// TwinCAT 3 PLC project MFX_BE_LENS_INTERLOCK
// ProgramVersion: 3.1.0.9
// libraries:
//   Tc2_Standard, * (Beckhoff Automation GmbH)
//   Tc2_System, * (Beckhoff Automation GmbH)
//   Tc3_Interfaces, * (Beckhoff Automation GmbH)
//   Tc3_Module, * (Beckhoff Automation GmbH)
//   Tc2_ModbusSrv,3.3.1.0,Beckhoff Automation GmbH
// project tree:
//   DUTs/ LENS.TcDUT, RADII_LIMIT.TcDUT, ST_FloatRange.TcDUT, ST_TableRow.TcDUT
//   / GlobalTextList.TcGTLO, PlcTask.TcTTO
//   GVLs/ GVL.TcGVL
//   POUs/ FB_EnergyTables.TcPOU, FB_LENS_SYSTEM.TcPOU, F_EFF_RADIUS.TcPOU, FB_HEARTBEAT.TcPOU (not stored), FB_LimitLookup.TcPOU, F_GetXRTLensIndex.TcPOU, MAIN.TcPOU, p_MPSSup.TcPOU, p_XLegacyPLCModbus.TcPOU (not stored)
//   POUs/Modbus/ p_ModbusRx_OutputCoils.TcPOU, p_ModbusRx_PLCMemory.TcPOU, p_ModbusTx_InputCoils.TcPOU, p_ModbusTx_InputReg.TcPOU, p_ModbusTx_OutputCoils.TcPOU, p_ModbusTx_PLCMemory.TcPOU
// real-time tasks:
//   TASK PlcTask: cycle T#10ms, priority 20, ADS port 350
// I/O:
//   DEVICE Device 2 (CX-BK)
//     Box 1 (CX-BK)
// variable links:
//   MFX_BE_LENS_INTERLOCK/MFX_BE_LENS_INTERLOCK Instance <-> Device 2 (CX-BK)/Box 1 (CX-BK)
//     PlcTask Outputs/GVL.bTRIP_MPS <-> Term 2 (KL2794)/Channel 1/Output

CONFIGURATION MFX_BE_LENS_INTERLOCK
    RESOURCE PLC ON TwinCAT3
        TASK PlcTask(INTERVAL := T#10ms, PRIORITY := 20);
        PROGRAM MAIN WITH PlcTask : MAIN;
    END_RESOURCE
END_CONFIGURATION

// ---- DUTs/LENS.TcDUT
TYPE LENS :
STRUCT
    IN     : BOOL; //Inserted state of the Lens
    KNOWN  : BOOL; //Whether state of Lens is definite
    RADIUS : REAL; //Current radius of lens
END_STRUCT
END_TYPE

// ---- DUTs/RADII_LIMIT.TcDUT
TYPE RADII_LIMIT :
STRUCT
    // Trip occurs when the effective radius falls inbetween TRIP_LOW and TRIP_HIGH (inclusive).
    TRIP_LOW  : REAL := 0;     // Trip effective radius low
    TRIP_HIGH : REAL := 10000; // Trip effective radius high
END_STRUCT
END_TYPE

// ---- DUTs/ST_FloatRange.TcDUT
TYPE ST_FloatRange :
STRUCT
    fLow  : REAL;
    fHigh : REAL;
END_STRUCT
END_TYPE

// ---- DUTs/ST_TableRow.TcDUT
TYPE ST_TableRow :
STRUCT
	fEnergy : LREAL;
    fLow  : LREAL;
    fHigh : LREAL;
END_STRUCT
END_TYPE

// ---- GVLs/GVL.TcGVL
VAR_GLOBAL
	(* Fault handling - inputs *)
    i_xFAULT_CLEAR    			: BOOL;  // Clear fault bit
	i_iUpdateRequestSeq			: DINT;  // Parameter update request sequence number

    (* Fault Handling - active faults *)
    bHeartbeatAlive     		: BOOL; // [Active] Whether heartbeat has updated
    bFAULT    AT %Q*    		: BOOL; // [Active] Whether Lens Interlock has tripped
    bStateFault	        		: BOOL; // [Active] Whether lens is in an unknown state
    bLimitSummaryFault			: BOOL; // [Active] Whether limit has been violated
    bTableLimitFault 			: BOOL;	// [Active] Energy/lens combination disallowed in table
    bMinEnergyFault 			: BOOL;	// [Active] Minimum energy not met
    bRequiresTransfocatorFault 	: BOOL; // [Active] Transfocator lens required to be inserted 

    (* Fault Handling - latched faults *)
	q_bHeartbeatLatch					: BOOL; // Latch: heartbeat fault
	q_bFaultLatch  						: BOOL; // Latch: summary for *any* fault
    q_bStateLatch 						: BOOL;	// Latch: motor state/position unknown 
    q_bLimitSummaryFaultLatch    		: BOOL; // Latch: Summary fault due to energy/lens combination
	q_bTableLimitFaultLatch 			: BOOL;	// Latch: Table disallowed range match
    q_bMinEnergyFaultLatch 				: BOOL; // Latch: Minimum energy not met
    q_bRequiresTransfocatorFaultLatch 	: BOOL; // Latch: Transfocator lens required to be inserted

	fbEnergyTables : FB_EnergyTables;
	
	(* Fault handling - MPS signals *)
    bTRIP_MPS AT %Q*    		: BOOL;  // [Active] Bit output to MPS (trip when LOW)
	
    (*Lens Information *)
    ////////////////////////////////
    XRT_LENSES : ARRAY[1..10] OF LENS; //Set of XRT Lenses
    TFS_LENSES : ARRAY[1..10] OF LENS; //Set of TFS Lenses
    XRT_RADIUS : REAL; //Current Radius of XRT lenses
    TFS_RADIUS : REAL; //Current Radius of TFS lenses
	
    XRT_LENS_SYSTEM : FB_LENS_SYSTEM;
    TFS_LENS_SYSTEM : FB_LENS_SYSTEM;

    (* Effective radius trip regions - per XRT lens configuration *)
    ////////////////////////////////////////////////////////////////
    NO_LENS_LIMIT : RADII_LIMIT;
    LENS1_LIMIT : RADII_LIMIT;
    LENS2_LIMIT : RADII_LIMIT;
    LENS3_LIMIT : RADII_LIMIT;	
	
	(* Feedback to the IOC *)
    q_stActiveLimit : RADII_LIMIT;
	
    fMinEnergies : ARRAY[0..3] OF LREAL;
    afbRequiresLensEnergyRange : ARRAY[0..3] OF ST_FloatRange;

    (* Heartbeat *)
    ////////////////////////////////
    i_xIOC_HEARTBEAT: BOOL; //Current status of heartbeat
    i_fPhotonEnergy : REAL; // Current photon energy (keep REAL for modbus compatibility)

    (* Modbus *)
    ///////////////////////////////
    LOTO_Override: BOOL := TRUE;
    /// test mb_Input_Coils[0] with "modpoll -r 32769 -t 1 127.0.0.1"
    mb_Input_Coils: ARRAY[0..255] OF BOOL;
    /// test mb_Output_Coils[0] with "modpoll -r 32769 -t 0 127.0.0.1"
    mb_Output_Coils: ARRAY[0..255] OF BOOL;
    /// test mb_Input_Registers[0] with "modpoll -r 32769 -t 3 127.0.0.1"
    mb_Input_Registers: ARRAY[0..255] OF WORD;
    /// test mb_Output_Registers[0] with "modpoll -r 32769 -t 4 127.0.0.1"
    mb_Output_Registers: ARRAY[0..255] OF WORD;
    /// test mb_PLC_Memory[0] with "modpoll -r 12289 -t 4 127.0.0.1"
    mb_PLC_Memory AT %MW0: ARRAY[0..1000] OF WORD;
	iCycleCount : WORD;

END_VAR

// ---- POUs/MAIN.TcPOU
PROGRAM MAIN
VAR
END_VAR

(* 16-bit cycle counter *)
iCycleCount := iCycleCount + 1;

fbEnergyTables();

(*  EPICS Rx UPDATE
    Modbus receive
*)
p_ModbusRx_OutputCoils();
p_ModbusRx_PLCMemory();
p_XLegacyPLCModbus();

(* Hard-code Lens Radii (microns) *)
XRT_LENSES[1].RADIUS := 750.0;
XRT_LENSES[2].RADIUS := 428.6;
XRT_LENSES[3].RADIUS := 333.3;

TFS_LENSES[1].RADIUS  := 0.0;   // A pinhole, not a lens.
TFS_LENSES[2].RADIUS  := 500.0;
TFS_LENSES[3].RADIUS  := 300.0;
TFS_LENSES[4].RADIUS  := 250.0;
TFS_LENSES[5].RADIUS  := 200.0;
TFS_LENSES[6].RADIUS  := 125.0;
TFS_LENSES[7].RADIUS  := 62.5;
TFS_LENSES[8].RADIUS  := 50.0;
TFS_LENSES[9].RADIUS  := 50.0;
TFS_LENSES[10].RADIUS := 50.0;

(* Additional trip settings

    Pre-focus 	Minimum energy [keV] 	Requires transfocator lens low [keV] 	Requires transfocator lens high [keV]
    NO_LENS 	0 	n/a 	n/a
    LENS3_333 	9.5 	9.5 	11.11
    LENS2_428 	8.28 	8.28 	10.02
    LENS1_750 	5.96 	5.96 	8.02

*)
fMinEnergies[0] := 0.0; (* No XRT lens *)
fMinEnergies[1] := 9500.0; (* XRT Lens 1 *)
fMinEnergies[2] := 8280.0; (* XRT lens 2 *)
fMinEnergies[3] := 5960.0; (* XRT lens 3 *)

afbRequiresLensEnergyRange[0].fLow := 0.0; (* No XRT lens / no restriction*)
afbRequiresLensEnergyRange[0].fHigh := 0.0;

afbRequiresLensEnergyRange[1].fLow := 9500.0; (* Lens 1: 9.5~11.11keV *)
afbRequiresLensEnergyRange[1].fHigh := 11110.0;

afbRequiresLensEnergyRange[2].fLow := 8280.0; (* Lens 2: 8.28 ~ 10.02 keV *)
afbRequiresLensEnergyRange[2].fHigh := 10020.0;

afbRequiresLensEnergyRange[3].fLow := 5960.0; (* Lens 3: 5.96 ~ 8.02 keV *)
afbRequiresLensEnergyRange[3].fHigh := 8020.0;

(*  MPS LOGIC SUMMARY *)
p_MPSSup();

(* 	EPICS Tx UPDATE
    Modbus Map Report
    IMPORTANT: This is the LAST subroutine to be called.
*)
p_ModbusTx_InputCoils();
p_ModbusTx_InputReg();
p_ModbusTx_PLCMemory();

END_PROGRAM

// ---- POUs/Modbus/p_ModbusRx_OutputCoils.TcPOU
PROGRAM p_ModbusRx_OutputCoils
VAR

END_VAR

//mb_Output_Coils[0];  //System Controls
//System Controls
//mb_Output_Coils[2];  //System Controls
//mb_Output_Coils[3];  //System Controls
//mb_Output_Coils[4];  //System Controls
//mb_Output_Coils[5];  //System Controls
//mb_Output_Coils[6];  //System Controls
//mb_Output_Coils[7];  //System Controls
//mb_Output_Coils[8];  //System Controls
//mb_Output_Coils[9];  //System Controls
TFS_LENSES[01].KNOWN:=TRUE;  //LOCKED OUT
TFS_LENSES[02].KNOWN:=mb_Output_Coils[11];  //Valve switch controls
TFS_LENSES[03].KNOWN:=mb_Output_Coils[12];  //Valve switch controls
TFS_LENSES[04].KNOWN:=mb_Output_Coils[13];  //Valve switch controls
TFS_LENSES[05].KNOWN:=mb_Output_Coils[14];  //Valve switch controls
TFS_LENSES[06].KNOWN:=mb_Output_Coils[15];  //Valve switch controls
TFS_LENSES[07].KNOWN:=mb_Output_Coils[16];  //Valve switch controls
TFS_LENSES[08].KNOWN:=mb_Output_Coils[17];  //Valve switch controls
TFS_LENSES[09].KNOWN:=mb_Output_Coils[18];  //Valve switch controls
TFS_LENSES[10].KNOWN:=mb_Output_Coils[19];  //Valve switch controls
XRT_LENSES[01].KNOWN:=mb_Output_Coils[20];
XRT_LENSES[02].KNOWN:=mb_Output_Coils[21];
XRT_LENSES[03].KNOWN:=mb_Output_Coils[22];
//mb_Output_Coils[23];  //Valve switch controls
//mb_Output_Coils[24];  //Valve switch controls
//mb_Output_Coils[25];  //Valve switch controls
//mb_Output_Coils[26];  //Valve switch controls
//mb_Output_Coils[27];  //Valve switch controls
//mb_Output_Coils[28];  //Valve switch controls
//mb_Output_Coils[29];  //Valve switch controls
TFS_LENSES[01].IN:=FALSE;  //Lockout
TFS_LENSES[02].IN:=mb_Output_Coils[31];  //Valve switch controls
TFS_LENSES[03].IN:=mb_Output_Coils[32];  //Valve switch controls
TFS_LENSES[04].IN:=mb_Output_Coils[33];  //Valve switch controls
TFS_LENSES[05].IN:=mb_Output_Coils[34];  //Valve switch controls
TFS_LENSES[06].IN:=mb_Output_Coils[35];  //Valve switch controls
TFS_LENSES[07].IN:=mb_Output_Coils[36];  //Valve switch controls
TFS_LENSES[08].IN:=mb_Output_Coils[37];  //Valve switch controls
TFS_LENSES[09].IN:=mb_Output_Coils[38];  //Valve switch controls
TFS_LENSES[10].IN:=mb_Output_Coils[39];  //Valve switch controls
XRT_LENSES[01].IN:=mb_Output_Coils[40];
XRT_LENSES[02].IN:=mb_Output_Coils[41];
XRT_LENSES[03].IN:=mb_Output_Coils[42];
//mb_Output_Coils[43];
//mb_Output_Coils[44];
//mb_Output_Coils[45];
//mb_Output_Coils[46];
//mb_Output_Coils[47];
//mb_Output_Coils[48];
//mb_Output_Coils[49];
i_xIOC_HEARTBEAT:=mb_Output_Coils[50];
i_xFAULT_CLEAR  :=mb_Output_Coils[51];
//mb_Output_Coils[52];  //Valve switch controls
//mb_Output_Coils[53];  //Valve switch controls
//mb_Output_Coils[54];  //Valve switch controls
//mb_Output_Coils[55];  //Valve switch controls
//mb_Output_Coils[56];  //Valve switch controls
//mb_Output_Coils[57];  //Valve switch controls
//mb_Output_Coils[58];  //Valve switch controls
//mb_Output_Coils[59];  //Valve switch controls
//mb_Output_Coils[60];  //Valve switch controls
//mb_Output_Coils[61];  //Valve switch controls
//mb_Output_Coils[62];  //Valve switch controls
//mb_Output_Coils[63];  //Valve switch controls
//mb_Output_Coils[64];  //Valve switch controls
//mb_Output_Coils[65];  //Valve switch controls
//mb_Output_Coils[66];  //Valve switch controls
//mb_Output_Coils[67];  //Valve switch controls
//mb_Output_Coils[68];  //Valve switch controls
//mb_Output_Coils[69];  //Valve switch controls
//mb_Output_Coils[70];  //Turbo Controls
//mb_Output_Coils[71];  //Turbo Controls
//mb_Output_Coils[72];  //Turbo Controls
//mb_Output_Coils[74];  //Turbo Controls
//mb_Output_Coils[75];  //Turbo Controls
//mb_Output_Coils[76];  //Turbo Controls
//mb_Output_Coils[77];  //Turbo Controls
//mb_Output_Coils[78];  //Turbo Controls
//mb_Output_Coils[79];  //Turbo Controls
//mb_Output_Coils[80];  //Turbo Controls
//mb_Output_Coils[81];  //Turbo Controls
//mb_Output_Coils[82];  //Turbo Controls
//mb_Output_Coils[83];  //Turbo Controls
//mb_Output_Coils[84];  //Turbo Controls
//mb_Output_Coils[85];  //Turbo Controls
//mb_Output_Coils[86];  //Turbo Controls
//mb_Output_Coils[87];  //Turbo Controls
//mb_Output_Coils[88];  //Turbo Controls
//mb_Output_Coils[89];  //Turbo Controls
//mb_Output_Coils[90];  //Turbo Controls
//mb_Output_Coils[91];  //Turbo Controls
//mb_Output_Coils[92];  //Turbo Controls
//mb_Output_Coils[93];  //Turbo Controls
//mb_Output_Coils[94];  //Turbo Controls
//mb_Output_Coils[95];  //Turbo Controls
//mb_Output_Coils[96];  //Turbo Controls
//mb_Output_Coils[97];  //Turbo Controls
//mb_Output_Coils[98];  //Turbo Controls
//mb_Output_Coils[99];  //Turbo Controls
//mb_Output_Coils[100];  //Turbo Controls
//mb_Output_Coils[101];  //Turbo Controls
//mb_Output_Coils[102];  //Turbo Controls
//mb_Output_Coils[103];  //Turbo Controls
//mb_Output_Coils[104];  //Turbo Controls
//mb_Output_Coils[105];  //Turbo Controls
//mb_Output_Coils[106];  //Turbo Controls
//mb_Output_Coils[107];  //Turbo Controls
//mb_Output_Coils[108];  //Turbo Controls
//mb_Output_Coils[109];  //Turbo Controls
//mb_Output_Coils[110];  //Turbo Controls
//mb_Output_Coils[111];  //Turbo Controls
//mb_Output_Coils[112];  //Turbo Controls
//mb_Output_Coils[113];  //Turbo Controls
//mb_Output_Coils[114];  //Turbo Controls
//mb_Output_Coils[115];  //Turbo Controls
//mb_Output_Coils[116];  //Turbo Controls
//mb_Output_Coils[117];  //Turbo Controls
//mb_Output_Coils[118];  //Turbo Controls
//mb_Output_Coils[119];  //Turbo Controls
//vgMXT_GCC_06.xHV_SW:=mb_Output_Coils[120];  //CC HV Enable
//vgDVD_GCC_02.xHV_SW:=mb_Output_Coils[121];  //CC HV Enable
//vgDVD_GCC_04.xHV_SW:=mb_Output_Coils[122];  //CC HV Enable
//vgMON_GCC_01.xHV_SW:=mb_Output_Coils[123];  //CC HV Enable
//vgDIA_GCC_01.xHV_SW:=mb_Output_Coils[124];  //CC HV Enable
//vgSB2_GCC_01.xHV_SW:=mb_Output_Coils[125];  //CC HV Enable
//vgDG1_GCC_01.xHV_SW:=mb_Output_Coils[126];  //CC HV Enable
//vgDG2_GCC_01.xHV_SW:=mb_Output_Coils[127];  //CC HV Enable
//mb_Output_Coils[128];  //CC HV Enable
//mb_Output_Coils[129];  //CC HV Enable
//mb_Output_Coils[130];  //CC HV Enable
//mb_Output_Coils[131];  //CC HV Enable
//mb_Output_Coils[132];  //CC HV Enable
//mb_Output_Coils[133];  //CC HV Enable
//mb_Output_Coils[134];  //CC HV Enable
//mb_Output_Coils[135];  //CC HV Enable
//mb_Output_Coils[136];  //CC HV Enable
//mb_Output_Coils[137];  //CC HV Enable
//mb_Output_Coils[138];  //CC HV Enable
//mb_Output_Coils[139];  //CC HV Enable
//mb_Output_Coils[140];  //CC HV Enable
//mb_Output_Coils[141];  //CC HV Enable
//mb_Output_Coils[142];  //CC HV Enable
//mb_Output_Coils[143];  //CC HV Enable
//mb_Output_Coils[144];  //CC HV Enable
//mb_Output_Coils[145];  //CC HV Enable
//mb_Output_Coils[146];  //CC HV Enable
//mb_Output_Coils[147];  //CC HV Enable
//mb_Output_Coils[148];  //CC HV Enable
//mb_Output_Coils[149];  //CC HV Enable
//mb_Output_Coils[150];  //CC HV Enable
//mb_Output_Coils[151];  //CC HV Enable
//mb_Output_Coils[152];  //CC HV Enable
//mb_Output_Coils[153];  //CC HV Enable
//mb_Output_Coils[154];  //CC HV Enable
//mb_Output_Coils[155];  //CC HV Enable
//mb_Output_Coils[156];  //CC HV Enable
//mb_Output_Coils[157];  //CC HV Enable
//mb_Output_Coils[158];  //CC HV Enable
//mb_Output_Coils[159];  //CC HV Enable
//mb_Output_Coils[160];  //
//mb_Output_Coils[161];  //
//mb_Output_Coils[162];  //
//mb_Output_Coils[163];  //
//mb_Output_Coils[164];  //
//mb_Output_Coils[165];  //
//mb_Output_Coils[166];  //
//mb_Output_Coils[167];  //
//mb_Output_Coils[168];  //
//mb_Output_Coils[169];  //
//mb_Output_Coils[170];  //
//mb_Output_Coils[171];  //
//mb_Output_Coils[172];  //
//mb_Output_Coils[173];  //
//mb_Output_Coils[174];  //
//mb_Output_Coils[175];  //
//mb_Output_Coils[176];  //
//mb_Output_Coils[177];  //
//mb_Output_Coils[178];  //
//mb_Output_Coils[179];  //
//mb_Output_Coils[180];  //
//mb_Output_Coils[181];  //
//mb_Output_Coils[182];  //
//mb_Output_Coils[183];  //
//mb_Output_Coils[184];  //
//mb_Output_Coils[185];  //
//mb_Output_Coils[186];  //
//mb_Output_Coils[187];  //
//mb_Output_Coils[188];  //
//mb_Output_Coils[189];  //
//mb_Output_Coils[190];  //
//mb_Output_Coils[191];  //
//mb_Output_Coils[192];  //
//mb_Output_Coils[193];  //
//mb_Output_Coils[194];  //
//mb_Output_Coils[195];  //
//mb_Output_Coils[196];  //
//mb_Output_Coils[197];  //
//mb_Output_Coils[198];  //
//mb_Output_Coils[199];  //
//mb_Output_Coils[200];  //Valve overrides
//mb_Output_Coils[201];  //Valve overrides
//mb_Output_Coils[202];  //Valve overrides
//mb_Output_Coils[203];  //Valve overrides
//mb_Output_Coils[204];  //
//mb_Output_Coils[205];  //
//mb_Output_Coils[206];  //
//mb_Output_Coils[207];  //
//mb_Output_Coils[208];  //
//mb_Output_Coils[209];  //
//mb_Output_Coils[210];  //
//mb_Output_Coils[211];  //
//mb_Output_Coils[212];  //
//mb_Output_Coils[213];  //
//mb_Output_Coils[214];  //
//mb_Output_Coils[215];  //
//mb_Output_Coils[216];  //
//mb_Output_Coils[217];  //
//mb_Output_Coils[218];  //
//mb_Output_Coils[219];  //
//mb_Output_Coils[220];  //
//mb_Output_Coils[221];  //
//mb_Output_Coils[222];  //
//mb_Output_Coils[223];  //
//mb_Output_Coils[224];  //
//mb_Output_Coils[225];  //
//mb_Output_Coils[226];  //
//mb_Output_Coils[227];  //
//mb_Output_Coils[228];  //
//mb_Output_Coils[229];  //
//mb_Output_Coils[230];  //
//mb_Output_Coils[231];  //
//mb_Output_Coils[232];  //
//mb_Output_Coils[233];  //
//mb_Output_Coils[234];  //
//mb_Output_Coils[235];  //
//mb_Output_Coils[236];  //
//mb_Output_Coils[237];  //
//mb_Output_Coils[238];  //
//mb_Output_Coils[239];  //
//mb_Output_Coils[240];  //
//mb_Output_Coils[241];  //
//mb_Output_Coils[242];  //
//mb_Output_Coils[243];  //
//mb_Output_Coils[244];  //
//mb_Output_Coils[245];  //
//mb_Output_Coils[246];  //
//mb_Output_Coils[247];  //
//mb_Output_Coils[248];  //
//mb_Output_Coils[249];  //
//mb_Output_Coils[250];  //
//mb_Output_Coils[251];  //
//mb_Output_Coils[252];  //
//mb_Output_Coils[253];  //
//mb_Output_Coils[254];  //
//mb_Output_Coils[255];  //

END_PROGRAM

// ---- POUs/Modbus/p_ModbusRx_PLCMemory.TcPOU
PROGRAM p_ModbusRx_PLCMemory
VAR
END_VAR

(*
{"MFX:LENS:",  "XRT_ONLY:LOW" , "aoFLOAT_PORT",    "0", "FLOAT32_LE",  "1", "1000",  "0", "um"}
{"MFX:LENS:",  "XRT_ONLY:HIGH", "aoFLOAT_PORT",    "2", "FLOAT32_LE",  "1", "1000",  "0", "um"}
{"MFX:LENS:", "LENS1_750:LOW" , "aoFLOAT_PORT",    "4", "FLOAT32_LE",  "1", "1000",  "0", "um"}
{"MFX:LENS:", "LENS1_750:HIGH", "aoFLOAT_PORT",    "6", "FLOAT32_LE",  "1", "1000",  "0", "um"}
{"MFX:LENS:", "LENS2_428:LOW" , "aoFLOAT_PORT",    "8", "FLOAT32_LE",  "1", "1000",  "0", "um"}
{"MFX:LENS:", "LENS2_428:HIGH", "aoFLOAT_PORT",   "10", "FLOAT32_LE",  "1", "1000",  "0", "um"}
{"MFX:LENS:", "LENS3_333:LOW" , "aoFLOAT_PORT",   "12", "FLOAT32_LE",  "1", "1000",  "0", "um"}
{"MFX:LENS:", "LENS3_333:HIGH", "aoFLOAT_PORT",   "14", "FLOAT32_LE",  "1", "1000",  "0", "um"}
*)
MEMCPY(srcAddr:=ADR(mb_PLC_Memory[ 0]), destAddr:=ADR(NO_LENS_LIMIT.TRIP_LOW), n:=SIZEOF(NO_LENS_LIMIT.TRIP_LOW));
MEMCPY(srcAddr:=ADR(mb_PLC_Memory[ 2]), destAddr:=ADR(NO_LENS_LIMIT.TRIP_HIGH), n:=SIZEOF(NO_LENS_LIMIT.TRIP_HIGH));

MEMCPY(srcAddr:=ADR(mb_PLC_Memory[ 4]), destAddr:=ADR(LENS1_LIMIT.TRIP_LOW), n:=SIZEOF(LENS1_LIMIT.TRIP_LOW));
MEMCPY(srcAddr:=ADR(mb_PLC_Memory[ 6]), destAddr:=ADR(LENS1_LIMIT.TRIP_HIGH), n:=SIZEOF(LENS1_LIMIT.TRIP_HIGH));

MEMCPY(srcAddr:=ADR(mb_PLC_Memory[ 8]), destAddr:=ADR(LENS2_LIMIT.TRIP_LOW), n:=SIZEOF(LENS2_LIMIT.TRIP_LOW));
MEMCPY(srcAddr:=ADR(mb_PLC_Memory[10]), destAddr:=ADR(LENS2_LIMIT.TRIP_HIGH), n:=SIZEOF(LENS2_LIMIT.TRIP_HIGH));

MEMCPY(srcAddr:=ADR(mb_PLC_Memory[12]), destAddr:=ADR(LENS3_LIMIT.TRIP_LOW), n:=SIZEOF(LENS3_LIMIT.TRIP_LOW));
MEMCPY(srcAddr:=ADR(mb_PLC_Memory[14]), destAddr:=ADR(LENS3_LIMIT.TRIP_HIGH), n:=SIZEOF(LENS3_LIMIT.TRIP_HIGH));

MEMCPY(srcAddr:=ADR(mb_PLC_Memory[16]), destAddr:=ADR(i_fPhotonEnergy), n:=SIZEOF(i_fPhotonEnergy));

MEMCPY(srcAddr:=ADR(mb_PLC_Memory[18]), destAddr:=ADR(i_iUpdateRequestSeq), n:=SIZEOF(i_iUpdateRequestSeq));

END_PROGRAM

// ---- POUs/p_MPSSup.TcPOU
PROGRAM p_MPSSup
VAR
    BEAT: FB_HEARTBEAT;
	fbHeartbeatLatch : RS;
	fbFaultLatch : RS;
    fbStateLatch : RS;
    fbLimitLatch : RS;
    fbTableLimitFaultLatch : RS;
    fbMinEnergyFaultLatch : RS;
    fbRequiresTransfocatorFaultLatch : RS;
	rtUpdate : R_TRIG;
	iLastSeq : DINT;
	bUpdateRequest: BOOL;
	
    LIMIT_FAULT : BOOL;

    fEnergyMin : LREAL;
    fRequiresTransfocatorEnergyLow : LREAL;
    fRequiresTransfocatorEnergyHigh : LREAL;
	fTripLow : LREAL;
	fTripHigh : LREAL;
	bEnergyInTable : BOOL;
	
    iLensIdx: INT;
	fbLimitLookup : FB_LimitLookup;

END_VAR

// Latch fault state
////////////////////

fbFaultLatch(SET:=bFAULT, RESET1:=i_xFAULT_CLEAR);
q_bFaultLatch := fbFaultLatch.Q1;

fbHeartbeatLatch(SET:=NOT bHeartbeatAlive, RESET1:=i_xFAULT_CLEAR);
q_bHeartbeatLatch := fbHeartbeatLatch.Q1;

fbStateLatch(SET:=bStateFault, RESET1:=i_xFAULT_CLEAR);
q_bStateLatch := fbStateLatch.Q1;

fbLimitLatch(SET:=bLimitSummaryFault, RESET1:=i_xFAULT_CLEAR);
q_bLimitSummaryFaultLatch := fbLimitLatch.Q1;

fbTableLimitFaultLatch(SET:=bTableLimitFault, RESET1:=i_xFAULT_CLEAR);
q_bTableLimitFaultLatch := fbTableLimitFaultLatch.Q1;

fbMinEnergyFaultLatch(SET:=bMinEnergyFault, RESET1:=i_xFAULT_CLEAR);
q_bMinEnergyFaultLatch := fbMinEnergyFaultLatch.Q1;

fbRequiresTransfocatorFaultLatch(SET:=bRequiresTransfocatorFault, RESET1:=i_xFAULT_CLEAR);
q_bRequiresTransfocatorFaultLatch := fbRequiresTransfocatorFaultLatch.Q1;

//IOC Heartbeat:
BEAT(BEAT:=i_xIOC_HEARTBEAT, DEADTIME:=TIME#0.5S);
bHeartbeatAlive := BEAT.ALIVE;

//XRT LENS SYSTEM
///////////////////////////
XRT_LENS_SYSTEM(LENSES:=XRT_LENSES, COUNT:=3);
XRT_RADIUS := XRT_LENS_SYSTEM.EFF_RADII; (* Propagated to EPICS *)

//TFS LENS SYSTEM
///////////////////////////
TFS_LENS_SYSTEM(LENSES:=TFS_LENSES, COUNT:=10);
TFS_RADIUS := TFS_LENS_SYSTEM.EFF_RADII; (* Propagated to EPICS *)

(* Reset our tracking variables *)
bTableLimitFault := FALSE;
bMinEnergyFault := FALSE;
bRequiresTransfocatorFault := FALSE;

(* Determine which XRT lens is inserted, and pick the correct range based on it. *)

IF NOT XRT_LENS_SYSTEM.UNKNOWN_FAULT THEN
	iLensIdx := F_GetXRTLensIndex();
	fbLimitLookup(
		fEnergy:=i_fPhotonEnergy,
		fLow=>fTripLow,
		fHigh=>fTripHigh,
		bEnergyInTable=>bEnergyInTable
	);

	q_stActiveLimit.TRIP_LOW := LREAL_TO_REAL(fTripLow);
	q_stActiveLimit.TRIP_HIGH := LREAL_TO_REAL(fTripHigh);

	IF bEnergyInTable AND fTripHigh > fTripLow THEN
		// Lens inserted and trip region specified:
		bTableLimitFault := (fTripLow <= TFS_RADIUS AND TFS_RADIUS <= fTripHigh);
	END_IF
	
	fEnergyMin := fMinEnergies[iLensIdx];
	fRequiresTransfocatorEnergyLow := afbRequiresLensEnergyRange[iLensIdx].fLow;
	fRequiresTransfocatorEnergyHigh := afbRequiresLensEnergyRange[iLensIdx].fHigh;
	
	(*
	Regardless of transfocator setting, the minimum energy must be
	greater than or equal to that shown in the table (Minimum energy [keV]).
	Trip if below.
	*)
	bMinEnergyFault := i_fPhotonEnergy < fEnergyMin;

	(*
	When a pre-focusing lens is inserted, there exists a range of photon
	energies in which at least one transfocator lens must be inserted.
	If the current photon energy is within this (inclusive) range and no
	lens is inserted, trip.
	*)
	IF fRequiresTransfocatorEnergyHigh > fRequiresTransfocatorEnergyLow THEN
		(* Check that we're in the given photon energy range *)
		IF fRequiresTransfocatorEnergyLow <= i_fPhotonEnergy AND i_fPhotonEnergy <= fRequiresTransfocatorEnergyHigh THEN
			(* And if so, trip when IN_COUNT == 0 *)
			bRequiresTransfocatorFault := (TFS_LENS_SYSTEM.IN_COUNT < 1);
		END_IF
	END_IF

END_IF

//Summarize faults
///////////////////////////

bLimitSummaryFault := (
	bTableLimitFault OR         // Inside the table-defined trip range
	bMinEnergyFault OR			// Below minimum required energy for XRT lens
	bRequiresTransfocatorFault	// Require transfocator lens in this range
);

//State Violations
bStateFault := (
	XRT_LENS_SYSTEM.UNKNOWN_FAULT OR  // XRT lens state unknown
	TFS_LENS_SYSTEM.UNKNOWN_FAULT OR  // Transfocator lens state unknown
	XRT_LENS_SYSTEM.IN_COUNT > 1      // Unexpected lens count
);

//Final Summary

// MPS trips when *LOW*. 
// 	So: bTRIP_MPS (False) when bFAULT (True)
// 	And bTRIP_MPS (True) when bFAULT (False)
bFAULT := bLimitSummaryFault OR bStateFault OR NOT bHeartbeatAlive;
bTRIP_MPS := NOT bFAULT;

(******************************)
(******************************)
(******************************)
(******************************)
bTRIP_MPS := TRUE; (* TEMPORARY: Alex requested the PLC never trip MPS for his overnight experiments *)
(* TODO: reviewers, this needs to be removed *)
(******************************)
(******************************)
(******************************)
(******************************)

END_PROGRAM

// ---- POUs/FB_LimitLookup.TcPOU
FUNCTION_BLOCK FB_LimitLookup
VAR_INPUT
	fEnergy : LREAL;
END_VAR
VAR_OUTPUT
	bEnergyInTable : BOOL;
	fLow : LREAL;
	fHigh : LREAL;
END_VAR
VAR
	(* TC version doesn't appear to support dynamic arrays here *)
	(* falling back to pointer-handling; sorry! *)
	stRow : POINTER TO ST_TableRow;
	stNextRow : POINTER TO ST_TableRow;
	iRowCount : UINT;
	iRowIdx : UINT;
	fSlope : LREAL;
	fEnergyDelta : LREAL;
	iLensIdx: INT;
END_VAR

iLensIdx := F_GetXRTLensIndex();

IF iLensIdx = 1 THEN
	stRow := ADR(fbEnergyTables.stLENS1_750);
	iRowCount := SIZEOF(fbEnergyTables.stLENS1_750) / SIZEOF(ST_TableRow);
ELSIF iLensIdx = 2 THEN
	stRow := ADR(fbEnergyTables.stLENS2_428);
	iRowCount := SIZEOF(fbEnergyTables.stLENS2_428) / SIZEOF(ST_TableRow);
ELSIF iLensIdx = 3 THEN
	stRow := ADR(fbEnergyTables.stLENS3_333);
	iRowCount := SIZEOF(fbEnergyTables.stLENS3_333) / SIZEOF(ST_TableRow);
ELSE
	stRow := ADR(fbEnergyTables.stNO_LENS);
	iRowCount := SIZEOF(fbEnergyTables.stNO_LENS) / SIZEOF(ST_TableRow);
END_IF

fLow := 0.0;
fHigh := 0.0;
bEnergyInTable := FALSE;

IF fEnergy < stRow^.fEnergy THEN
	RETURN;
END_IF

FOR iRowIdx := 0 TO iRowCount - 2
DO
(*
 result->energy = find_energy;
 double slope = (rows[upper_idx].low - rows[lower_idx].low) / delta_energy;
 result->low = rows[lower_idx].low + slope * (find_energy - rows[lower_idx].energy);

 slope = (rows[upper_idx].high - rows[lower_idx].high) / delta_energy;
 result->high = rows[lower_idx].high + slope * (find_energy - rows[lower_idx].energy);
*)
	stNextRow := ADR(stRow[1]);
	IF fEnergy >= stRow^.fEnergy AND fEnergy <= stNextRow^.fEnergy THEN
		fEnergyDelta := stNextRow^.fEnergy - stRow^.fEnergy;
		IF fEnergyDelta > 0.0 THEN
			bEnergyInTable := TRUE;
			// Interpolate between the points
			fSlope := (stNextRow^.fLow - stRow^.fLow) / fEnergyDelta;
			fLow := stRow^.fLow + fSlope * (fEnergy - stRow^.fEnergy);

			fSlope := (stNextRow^.fHigh - stRow^.fHigh) / fEnergyDelta;
			fHigh := stRow^.fHigh + fSlope * (fEnergy - stRow^.fEnergy);
		END_IF	
		RETURN;
	END_IF
	stRow := stNextRow;
END_FOR

END_FUNCTION_BLOCK

// ---- POUs/F_GetXRTLensIndex.TcPOU
FUNCTION F_GetXRTLensIndex : INT
VAR_INPUT
END_VAR
VAR
END_VAR

IF XRT_LENS_SYSTEM.LENSES[1].IN THEN
	F_GetXRTLensIndex := 1;
ELSIF XRT_LENS_SYSTEM.LENSES[2].IN THEN
	F_GetXRTLensIndex := 2;
ELSIF XRT_LENS_SYSTEM.LENSES[3].IN THEN
	F_GetXRTLensIndex := 3;
ELSE
	F_GetXRTLensIndex := 0;
END_IF

END_FUNCTION

// ---- POUs/Modbus/p_ModbusTx_InputCoils.TcPOU
PROGRAM p_ModbusTx_InputCoils
VAR
END_VAR
VAR_OUTPUT
END_VAR

(** NOTE: These values are mirrored in PLC memory output as well. **)
(** From an EPICS client perspective, it's easier to keep the data
    in synchronization when sent in one packet. The IOC now uses
    those values and these are vestigial for now.
**)


(* Online/active values *)
mb_Input_Coils[0]:=bHeartbeatAlive;
mb_Input_Coils[1]:=bFAULT;
mb_Input_Coils[2]:=bStateFault;
mb_Input_Coils[3]:=bLimitSummaryFault;
mb_Input_Coils[4]:=bMinEnergyFault;
mb_Input_Coils[5]:=bRequiresTransfocatorFault;
mb_Input_Coils[6]:=bTableLimitFault;
mb_Input_Coils[7]:=FALSE;
mb_Input_Coils[8]:=FALSE;
mb_Input_Coils[9]:=FALSE;

(* Latched fault information *)
mb_Input_Coils[10]:=q_bHeartbeatLatch;
mb_Input_Coils[11]:=q_bFaultLatch;
mb_Input_Coils[12]:=q_bStateLatch;
mb_Input_Coils[13]:=q_bLimitSummaryFaultLatch;
mb_Input_Coils[14]:=q_bMinEnergyFaultLatch;
mb_Input_Coils[15]:=q_bRequiresTransfocatorFaultLatch;
mb_Input_Coils[16]:=q_bTableLimitFaultLatch;
mb_Input_Coils[17]:=FALSE;
mb_Input_Coils[18]:=FALSE;
mb_Input_Coils[19]:=FALSE;

mb_Input_Coils[20]:=FALSE;  //Valve position readbacks
mb_Input_Coils[21]:=FALSE;  //Valve position readbacks
mb_Input_Coils[22]:=FALSE;  //Valve position readbacks
mb_Input_Coils[23]:=FALSE;  //Valve position readbacks
mb_Input_Coils[24]:=FALSE;  //Valve position readbacks
mb_Input_Coils[25]:=FALSE;  //Valve position readbacks
mb_Input_Coils[26]:=FALSE;  //Valve position readbacks
mb_Input_Coils[27]:=FALSE;  //Valve position readbacks
mb_Input_Coils[28]:=FALSE;  //Valve position readbacks
mb_Input_Coils[29]:=FALSE;  //Valve position readbacks
mb_Input_Coils[30]:=FALSE;  //Valve position readbacks
mb_Input_Coils[31]:=FALSE;  //Valve position readbacks
mb_Input_Coils[32]:=FALSE;  //Valve position readbacks
mb_Input_Coils[33]:=FALSE;  //Valve position readbacks
mb_Input_Coils[34]:=FALSE;  //Valve position readbacks
mb_Input_Coils[35]:=FALSE;  //Valve position readbacks
mb_Input_Coils[36]:=FALSE;  //Valve position readbacks
mb_Input_Coils[37]:=FALSE;  //Valve position readbacks
mb_Input_Coils[38]:=FALSE;  //Valve position readbacks
mb_Input_Coils[39]:=FALSE;  //Valve position readbacks
mb_Input_Coils[40]:=FALSE;  //Valve position readbacks
mb_Input_Coils[41]:=FALSE;  //Valve position readbacks
mb_Input_Coils[42]:=FALSE;  //Valve position readbacks
mb_Input_Coils[43]:=FALSE;  //Valve position readbacks
mb_Input_Coils[44]:=FALSE;  //Valve position readbacks
mb_Input_Coils[45]:=FALSE;  //Valve position readbacks
mb_Input_Coils[46]:=FALSE;  //Valve position readbacks
mb_Input_Coils[47]:=FALSE;  //Valve position readbacks
mb_Input_Coils[48]:=FALSE;  //Valve position readbacks
mb_Input_Coils[49]:=FALSE;  //Valve position readbacks
mb_Input_Coils[50]:=FALSE;  //Valve position readbacks
mb_Input_Coils[51]:=FALSE;  //Valve position readbacks
mb_Input_Coils[52]:=FALSE;  //Valve position readbacks
mb_Input_Coils[53]:=FALSE;  //Valve position readbacks
mb_Input_Coils[54]:=FALSE;  //Valve position readbacks
mb_Input_Coils[55]:=FALSE;  //Valve position readbacks
mb_Input_Coils[56]:=FALSE;  //Valve position readbacks
mb_Input_Coils[57]:=FALSE;  //Valve position readbacks
mb_Input_Coils[58]:=FALSE;  //Valve position readbacks
mb_Input_Coils[59]:=FALSE;  //Valve position readbacks
mb_Input_Coils[60]:=FALSE;  //Valve position readbacks
mb_Input_Coils[61]:=FALSE;  //Valve position readbacks
mb_Input_Coils[62]:=FALSE;  //Valve position readbacks
mb_Input_Coils[63]:=FALSE;  //Valve position readbacks
mb_Input_Coils[64]:=FALSE;  //Valve position readbacks
mb_Input_Coils[65]:=FALSE;  //Valve position readbacks
mb_Input_Coils[66]:=FALSE;  //Valve position readbacks
mb_Input_Coils[67]:=FALSE;  //Valve position readbacks
mb_Input_Coils[68]:=FALSE;  //Valve position readbacks
mb_Input_Coils[69]:=FALSE;  //Valve position readbacks
mb_Input_Coils[70]:=FALSE;  //Valve position readbacks
mb_Input_Coils[71]:=FALSE;  //Valve position readbacks
mb_Input_Coils[72]:=FALSE;  //Valve position readbacks
mb_Input_Coils[73]:=FALSE;  //Valve position readbacks
mb_Input_Coils[74]:=FALSE;  //Valve position readbacks
mb_Input_Coils[75]:=FALSE;  //Valve position readbacks
mb_Input_Coils[76]:=FALSE;  //Valve position readbacks
mb_Input_Coils[77]:=FALSE;  //Valve position readbacks
mb_Input_Coils[78]:=FALSE;  //Valve position readbacks
mb_Input_Coils[79]:=FALSE;  //Valve position readbacks
mb_Input_Coils[80]:=FALSE;  //Valve position readbacks
mb_Input_Coils[81]:=FALSE;  //Valve position readbacks
mb_Input_Coils[82]:=FALSE;  //Valve position readbacks
mb_Input_Coils[83]:=FALSE;  //Valve position readbacks
mb_Input_Coils[84]:=FALSE;  //Valve position readbacks
mb_Input_Coils[85]:=FALSE;  //Valve position readbacks
mb_Input_Coils[86]:=FALSE;  //Valve position readbacks
mb_Input_Coils[87]:=FALSE;  //Valve position readbacks
mb_Input_Coils[88]:=FALSE;  //Valve position readbacks
mb_Input_Coils[89]:=FALSE;  //Valve position readbacks
mb_Input_Coils[90]:=FALSE;  //Valve position readbacks
mb_Input_Coils[91]:=FALSE;  //Valve position readbacks
mb_Input_Coils[92]:=FALSE;  //Valve position readbacks
mb_Input_Coils[93]:=FALSE;  //Valve position readbacks
mb_Input_Coils[94]:=FALSE;  //Valve position readbacks
mb_Input_Coils[95]:=FALSE;  //Valve position readbacks
mb_Input_Coils[96]:=FALSE;  //Valve position readbacks
mb_Input_Coils[97]:=FALSE;  //Valve position readbacks
mb_Input_Coils[98]:=FALSE;  //Valve position readbacks
mb_Input_Coils[99]:=FALSE;  //Valve position readbacks
mb_Input_Coils[100]:=FALSE;  //Valve position readbacks
mb_Input_Coils[101]:=FALSE;  //Valve position readbacks
mb_Input_Coils[102]:=FALSE;  //Valve position readbacks
mb_Input_Coils[103]:=FALSE;  //Valve position readbacks
mb_Input_Coils[104]:=FALSE;  //Valve position readbacks
mb_Input_Coils[105]:=FALSE;  //Valve position readbacks
mb_Input_Coils[106]:=FALSE;  //Valve position readbacks
mb_Input_Coils[107]:=FALSE;  //Valve position readbacks
mb_Input_Coils[108]:=FALSE;  //Valve position readbacks
mb_Input_Coils[109]:=FALSE;  //Valve position readbacks
mb_Input_Coils[110]:=FALSE;  //Valve position readbacks
mb_Input_Coils[111]:=FALSE;  //Valve position readbacks
mb_Input_Coils[112]:=FALSE;  //Valve position readbacks
mb_Input_Coils[113]:=FALSE;  //Valve position readbacks
mb_Input_Coils[114]:=FALSE;  //Valve position readbacks
mb_Input_Coils[115]:=FALSE;  //Valve position readbacks
mb_Input_Coils[116]:=FALSE;  //Valve position readbacks
mb_Input_Coils[117]:=FALSE;  //Valve position readbacks
mb_Input_Coils[118]:=FALSE;  //Valve position readbacks
mb_Input_Coils[119]:=FALSE;  //Valve position readbacks
mb_Input_Coils[120]:=FALSE;  //Turbo pump readbacks
mb_Input_Coils[121]:=FALSE;  //Turbo pump readbacks
mb_Input_Coils[122]:=FALSE;  //Turbo pump readbacks
mb_Input_Coils[123]:=FALSE;  //Turbo pump readbacks
mb_Input_Coils[124]:=FALSE;  //Turbo pump readbacks
mb_Input_Coils[125]:=FALSE;  //Turbo pump readbacks
mb_Input_Coils[126]:=FALSE;  //Turbo pump readbacks
mb_Input_Coils[127]:=FALSE;  //Turbo pump readbacks
mb_Input_Coils[128]:=FALSE;  //Turbo pump readbacks
mb_Input_Coils[129]:=FALSE;  //Turbo pump readbacks
mb_Input_Coils[130]:=FALSE;  //Turbo pump readbacks
mb_Input_Coils[131]:=FALSE;  //Turbo pump readbacks
mb_Input_Coils[132]:=FALSE;  //Turbo pump readbacks
mb_Input_Coils[133]:=FALSE;  //Turbo pump readbacks
mb_Input_Coils[134]:=FALSE;  //Turbo pump readbacks
mb_Input_Coils[135]:=FALSE;  //Turbo pump readbacks
mb_Input_Coils[136]:=FALSE;  //Turbo pump readbacks
mb_Input_Coils[137]:=FALSE;  //Turbo pump readbacks
mb_Input_Coils[138]:=FALSE;  //Turbo pump readbacks
mb_Input_Coils[139]:=FALSE;  //Turbo pump readbacks
mb_Input_Coils[140]:=FALSE;  //Turbo pump readbacks
mb_Input_Coils[141]:=FALSE;  //Turbo pump readbacks
mb_Input_Coils[142]:=FALSE;  //Turbo pump readbacks
mb_Input_Coils[143]:=FALSE;  //Turbo pump readbacks
mb_Input_Coils[144]:=FALSE;  //Turbo pump readbacks
mb_Input_Coils[145]:=FALSE;  //Turbo pump readbacks
mb_Input_Coils[146]:=FALSE;  //Turbo pump readbacks
mb_Input_Coils[147]:=FALSE;  //Turbo pump readbacks
mb_Input_Coils[148]:=FALSE;  //Turbo pump readbacks
mb_Input_Coils[149]:=FALSE;  //Turbo pump readbacks
mb_Input_Coils[150]:=FALSE;  //Turbo pump readbacks
mb_Input_Coils[151]:=FALSE;  //Turbo pump readbacks
mb_Input_Coils[152]:=FALSE;  //Turbo pump readbacks
mb_Input_Coils[153]:=FALSE;  //Turbo pump readbacks
mb_Input_Coils[154]:=FALSE;  //Turbo pump readbacks
mb_Input_Coils[155]:=FALSE;  //Turbo pump readbacks
mb_Input_Coils[156]:=FALSE;  //Turbo pump readbacks
mb_Input_Coils[157]:=FALSE;  //Turbo pump readbacks
mb_Input_Coils[158]:=FALSE;  //Turbo pump readbacks
mb_Input_Coils[159]:=FALSE;  //Turbo pump readbacks
mb_Input_Coils[160]:=FALSE;  //Turbo pump readbacks
mb_Input_Coils[161]:=FALSE;  //Turbo pump readbacks
mb_Input_Coils[162]:=FALSE;  //Turbo pump readbacks
mb_Input_Coils[163]:=FALSE;  //Turbo pump readbacks
mb_Input_Coils[164]:=FALSE;  //Turbo pump readbacks
mb_Input_Coils[165]:=FALSE;  //Turbo pump readbacks
mb_Input_Coils[166]:=FALSE;  //Turbo pump readbacks
mb_Input_Coils[167]:=FALSE;  //Turbo pump readbacks
mb_Input_Coils[168]:=FALSE;  //Turbo pump readbacks
mb_Input_Coils[169]:=FALSE;  //Turbo pump readbacks
mb_Input_Coils[170]:=FALSE;  //Turbo pump readbacks
mb_Input_Coils[171]:=FALSE;  //Turbo pump readbacks
mb_Input_Coils[172]:=FALSE;  //Turbo pump readbacks
mb_Input_Coils[173]:=FALSE;  //Turbo pump readbacks
mb_Input_Coils[174]:=FALSE;  //Turbo pump readbacks
mb_Input_Coils[175]:=FALSE;  //Turbo pump readbacks
mb_Input_Coils[176]:=FALSE;  //Turbo pump readbacks
mb_Input_Coils[177]:=FALSE;  //Turbo pump readbacks
mb_Input_Coils[178]:=FALSE;  //Turbo pump readbacks
mb_Input_Coils[179]:=FALSE;  //Turbo pump readbacks
mb_Input_Coils[180]:=FALSE;  //Turbo pump readbacks
mb_Input_Coils[181]:=FALSE;  //Turbo pump readbacks
mb_Input_Coils[182]:=FALSE;  //Turbo pump readbacks
mb_Input_Coils[183]:=FALSE;  //Turbo pump readbacks
mb_Input_Coils[184]:=FALSE;  //Turbo pump readbacks
mb_Input_Coils[185]:=FALSE;  //Turbo pump readbacks
mb_Input_Coils[186]:=FALSE;  //Turbo pump readbacks
mb_Input_Coils[187]:=FALSE;  //Turbo pump readbacks
mb_Input_Coils[188]:=FALSE;  //Turbo pump readbacks
mb_Input_Coils[189]:=FALSE;  //Turbo pump readbacks
mb_Input_Coils[190]:=FALSE;  //Turbo pump readbacks
mb_Input_Coils[191]:=FALSE;  //Turbo pump readbacks
mb_Input_Coils[192]:=FALSE;  //Turbo pump readbacks
mb_Input_Coils[193]:=FALSE;  //Turbo pump readbacks
mb_Input_Coils[194]:=FALSE;  //Turbo pump readbacks
mb_Input_Coils[195]:=FALSE;  //Turbo pump readbacks
mb_Input_Coils[196]:=FALSE;  //Turbo pump readbacks
mb_Input_Coils[197]:=FALSE;  //Turbo pump readbacks
mb_Input_Coils[198]:=FALSE;  //Turbo pump readbacks
mb_Input_Coils[199]:=FALSE;  //Turbo pump readbacks
mb_Input_Coils[200]:=FALSE;  //Turbo pump readbacks
mb_Input_Coils[201]:=FALSE;  //Turbo pump readbacks
mb_Input_Coils[202]:=FALSE;  //Turbo pump readbacks
mb_Input_Coils[203]:=FALSE;  //Turbo pump readbacks
mb_Input_Coils[204]:=FALSE;  //Turbo pump readbacks
mb_Input_Coils[205]:=FALSE;  //Turbo pump readbacks
mb_Input_Coils[206]:=FALSE;  //Turbo pump readbacks
mb_Input_Coils[207]:=FALSE;  //Turbo pump readbacks
mb_Input_Coils[208]:=FALSE;  //Turbo pump readbacks
mb_Input_Coils[209]:=FALSE;  //Turbo pump readbacks
mb_Input_Coils[210]:=FALSE;  //Turbo pump readbacks
mb_Input_Coils[211]:=FALSE;  //Turbo pump readbacks
mb_Input_Coils[212]:=FALSE;  //Turbo pump readbacks
mb_Input_Coils[213]:=FALSE;  //Turbo pump readbacks
mb_Input_Coils[214]:=FALSE;  //Turbo pump readbacks
mb_Input_Coils[215]:=FALSE;  //Turbo pump readbacks
mb_Input_Coils[216]:=FALSE;  //Turbo pump readbacks
mb_Input_Coils[217]:=FALSE;  //Turbo pump readbacks
mb_Input_Coils[218]:=FALSE;  //Turbo pump readbacks
mb_Input_Coils[219]:=FALSE;  //Turbo pump readbacks
mb_Input_Coils[220]:=FALSE;  //VG readbacks
mb_Input_Coils[221]:=FALSE;  //VG readbacks
mb_Input_Coils[222]:=FALSE;  //VG readbacks
mb_Input_Coils[223]:=FALSE;  //VG readbacks
mb_Input_Coils[224]:=FALSE;  //VG readbacks
mb_Input_Coils[225]:=FALSE;  //VG readbacks
mb_Input_Coils[226]:=FALSE;  //VG readbacks
mb_Input_Coils[227]:=FALSE;  //VG readbacks
mb_Input_Coils[228]:=FALSE;  //VG readbacks
mb_Input_Coils[229]:=FALSE;  //VG readbacks
mb_Input_Coils[230]:=FALSE;  //VG readbacks
mb_Input_Coils[231]:=FALSE;  //VG readbacks
mb_Input_Coils[232]:=FALSE;  //VG readbacks
mb_Input_Coils[233]:=FALSE;  //VG readbacks
mb_Input_Coils[234]:=FALSE;  //VG readbacks
mb_Input_Coils[235]:=FALSE;  //VG readbacks
mb_Input_Coils[236]:=FALSE;  //VG readbacks
mb_Input_Coils[237]:=FALSE;  //VG readbacks
mb_Input_Coils[238]:=FALSE;  //VG readbacks
mb_Input_Coils[239]:=FALSE;  //VG readbacks
mb_Input_Coils[240]:=FALSE;  //VG readbacks
mb_Input_Coils[241]:=FALSE;  //VG readbacks
mb_Input_Coils[242]:=FALSE;  //VG readbacks
mb_Input_Coils[243]:=FALSE;  //VG readbacks
mb_Input_Coils[244]:=FALSE;  //VG readbacks
mb_Input_Coils[245]:=FALSE;  //VG readbacks
mb_Input_Coils[246]:=FALSE;  //VG readbacks
mb_Input_Coils[247]:=FALSE;  //VG readbacks
mb_Input_Coils[248]:=FALSE;  //VG readbacks
mb_Input_Coils[249]:=FALSE;  //VG readbacks
mb_Input_Coils[250]:=FALSE;  //VG readbacks
mb_Input_Coils[251]:=FALSE;  //VG readbacks
mb_Input_Coils[252]:=FALSE;  //VG readbacks
mb_Input_Coils[253]:=FALSE;  //VG readbacks
mb_Input_Coils[254]:=FALSE;  //VG readbacks
mb_Input_Coils[255]:=FALSE;  //VG readbacks

END_PROGRAM

// ---- POUs/Modbus/p_ModbusTx_InputReg.TcPOU
PROGRAM p_ModbusTx_InputReg
VAR

END_VAR

mb_Input_Registers[0]:=0;  //System info
mb_Input_Registers[1]:=0;  //System info
mb_Input_Registers[2]:=0;  //System info
mb_Input_Registers[3]:=0;  //System info
mb_Input_Registers[4]:=0;  //System info
mb_Input_Registers[5]:=0;  //System info
mb_Input_Registers[6]:=0;  //System info
mb_Input_Registers[7]:=0;  //System info
mb_Input_Registers[8]:=0;  //System info
mb_Input_Registers[9]:=0;  //System info
mb_Input_Registers[10]:=0;  //VG pressure readbacks
mb_Input_Registers[11]:=0;  //VG pressure readbacks
mb_Input_Registers[12]:=0;  //VG pressure readbacks
mb_Input_Registers[13]:=0;  //VG pressure readbacks
mb_Input_Registers[14]:=0;  //VG pressure readbacks
mb_Input_Registers[15]:=0;  //VG pressure readbacks
mb_Input_Registers[16]:=0;  //VG pressure readbacks
mb_Input_Registers[17]:=0;  //VG pressure readbacks
mb_Input_Registers[18]:=0;  //VG pressure readbacks
mb_Input_Registers[19]:=0;  //VG pressure readbacks
mb_Input_Registers[20]:=0;  //VG pressure readbacks
mb_Input_Registers[21]:=0;  //VG pressure readbacks
mb_Input_Registers[22]:=0;  //VG pressure readbacks
mb_Input_Registers[23]:=0;  //VG pressure readbacks
mb_Input_Registers[24]:=0;  //VG pressure readbacks
mb_Input_Registers[25]:=0;  //VG pressure readbacks
mb_Input_Registers[26]:=0;  //VG pressure readbacks
mb_Input_Registers[27]:=0;  //VG pressure readbacks
mb_Input_Registers[28]:=0;  //VG pressure readbacks
mb_Input_Registers[29]:=0;  //VG pressure readbacks
mb_Input_Registers[30]:=0;  //VG pressure readbacks
mb_Input_Registers[31]:=0;  //VG pressure readbacks
mb_Input_Registers[32]:=0;  //VG pressure readbacks
mb_Input_Registers[33]:=0;  //VG pressure readbacks
mb_Input_Registers[34]:=0;  //VG pressure readbacks
mb_Input_Registers[35]:=0;  //VG pressure readbacks
mb_Input_Registers[36]:=0;  //VG pressure readbacks
mb_Input_Registers[37]:=0;  //VG pressure readbacks
mb_Input_Registers[38]:=0;  //VG pressure readbacks
mb_Input_Registers[39]:=0;  //VG pressure readbacks
mb_Input_Registers[40]:=0;  //VG pressure readbacks
mb_Input_Registers[41]:=0;  //VG pressure readbacks
mb_Input_Registers[42]:=0;  //VG pressure readbacks
mb_Input_Registers[43]:=0;  //VG pressure readbacks
mb_Input_Registers[44]:=0;  //VG pressure readbacks
mb_Input_Registers[45]:=0;  //VG pressure readbacks
mb_Input_Registers[46]:=0;  //VG pressure readbacks
mb_Input_Registers[47]:=0;  //VG pressure readbacks
mb_Input_Registers[48]:=0;  //VG pressure readbacks
mb_Input_Registers[49]:=0;  //VG pressure readbacks
mb_Input_Registers[50]:=0;  //VG pressure readbacks
mb_Input_Registers[51]:=0;  //VG pressure readbacks
mb_Input_Registers[52]:=0;  //VG pressure readbacks
mb_Input_Registers[53]:=0;  //VG pressure readbacks
mb_Input_Registers[54]:=0;  //VG pressure readbacks
mb_Input_Registers[55]:=0;  //VG pressure readbacks
mb_Input_Registers[56]:=0;  //VG pressure readbacks
mb_Input_Registers[57]:=0;  //VG pressure readbacks
mb_Input_Registers[58]:=0;  //VG pressure readbacks
mb_Input_Registers[59]:=0;  //VG pressure readbacks
mb_Input_Registers[60]:=0;  //VG pressure readbacks
mb_Input_Registers[61]:=0;  //VG pressure readbacks
mb_Input_Registers[62]:=0;  //VG pressure readbacks
mb_Input_Registers[63]:=0;  //VG pressure readbacks
mb_Input_Registers[64]:=0;  //VG pressure readbacks
mb_Input_Registers[65]:=0;  //VG pressure readbacks
mb_Input_Registers[66]:=0;  //VG pressure readbacks
mb_Input_Registers[67]:=0;  //VG pressure readbacks
mb_Input_Registers[68]:=0;  //VG pressure readbacks
mb_Input_Registers[69]:=0;  //VG pressure readbacks
mb_Input_Registers[70]:=0;  //VG state readbacks
mb_Input_Registers[71]:=0;  //VG state readbacks
mb_Input_Registers[72]:=0;  //VG state readbacks
mb_Input_Registers[73]:=0;  //VG state readbacks
mb_Input_Registers[74]:=0;  //VG state readbacks
mb_Input_Registers[75]:=0;  //VG state readbacks
mb_Input_Registers[76]:=0;  //VG state readbacks
mb_Input_Registers[77]:=0;  //VG state readbacks
mb_Input_Registers[78]:=0;  //VG state readbacks
mb_Input_Registers[79]:=0;  //VG state readbacks
mb_Input_Registers[80]:=0;  //VG state readbacks
mb_Input_Registers[81]:=0;  //VG state readbacks
mb_Input_Registers[82]:=0;  //VG state readbacks
mb_Input_Registers[83]:=0;  //VG state readbacks
mb_Input_Registers[84]:=0;  //VG state readbacks
mb_Input_Registers[85]:=0;  //VG state readbacks
mb_Input_Registers[86]:=0;  //VG state readbacks
mb_Input_Registers[87]:=0;  //VG state readbacks
mb_Input_Registers[88]:=0;  //VG state readbacks
mb_Input_Registers[89]:=0;  //VG state readbacks
mb_Input_Registers[90]:=0;  //VG state readbacks
mb_Input_Registers[91]:=0;  //VG state readbacks
mb_Input_Registers[92]:=0;  //VG state readbacks
mb_Input_Registers[93]:=0;  //VG state readbacks
mb_Input_Registers[94]:=0;  //VG state readbacks
mb_Input_Registers[95]:=0;  //VG state readbacks
mb_Input_Registers[96]:=0;  //VG state readbacks
mb_Input_Registers[97]:=0;  //VG state readbacks
mb_Input_Registers[98]:=0;  //VG state readbacks
mb_Input_Registers[99]:=0;  //VG state readbacks
mb_Input_Registers[100]:=0;  //VG state readbacks
mb_Input_Registers[101]:=0;  //VG state readbacks
mb_Input_Registers[102]:=0;  //VG state readbacks
mb_Input_Registers[103]:=0;  //VG state readbacks
mb_Input_Registers[104]:=0;  //VG state readbacks
mb_Input_Registers[105]:=0;  //VG state readbacks
mb_Input_Registers[106]:=0;  //VG state readbacks
mb_Input_Registers[107]:=0;  //VG state readbacks
mb_Input_Registers[108]:=0;  //VG state readbacks
mb_Input_Registers[109]:=0;  //VG state readbacks
mb_Input_Registers[110]:=0;  //VG state readbacks
mb_Input_Registers[111]:=0;  //VG state readbacks
mb_Input_Registers[112]:=0;  //VG state readbacks
mb_Input_Registers[113]:=0;  //VG state readbacks
mb_Input_Registers[114]:=0;  //VG state readbacks
mb_Input_Registers[115]:=0;  //VG state readbacks
mb_Input_Registers[116]:=0;  //VG state readbacks
mb_Input_Registers[117]:=0;  //VG state readbacks
mb_Input_Registers[118]:=0;  //VG state readbacks
mb_Input_Registers[119]:=0;  //VG state readbacks
mb_Input_Registers[120]:=0;  //default
mb_Input_Registers[121]:=0;  //default
mb_Input_Registers[122]:=0;  //default
mb_Input_Registers[123]:=0;  //default
mb_Input_Registers[124]:=0;  //default
mb_Input_Registers[125]:=0;  //default
mb_Input_Registers[126]:=0;  //default
mb_Input_Registers[127]:=0;  //default
mb_Input_Registers[128]:=0;  //default
mb_Input_Registers[129]:=0;  //default
mb_Input_Registers[130]:=0;  //default
mb_Input_Registers[131]:=0;  //default
mb_Input_Registers[132]:=0;  //default
mb_Input_Registers[133]:=0;  //default
mb_Input_Registers[134]:=0;  //default
mb_Input_Registers[135]:=0;  //default
mb_Input_Registers[136]:=0;  //default
mb_Input_Registers[137]:=0;  //default
mb_Input_Registers[138]:=0;  //default
mb_Input_Registers[139]:=0;  //default
mb_Input_Registers[140]:=0;  //default
mb_Input_Registers[141]:=0;  //default
mb_Input_Registers[142]:=0;  //default
mb_Input_Registers[143]:=0;  //default
mb_Input_Registers[144]:=0;  //default
mb_Input_Registers[145]:=0;  //default
mb_Input_Registers[146]:=0;  //default
mb_Input_Registers[147]:=0;  //default
mb_Input_Registers[148]:=0;  //default
mb_Input_Registers[149]:=0;  //default
mb_Input_Registers[150]:=0;  //default
mb_Input_Registers[151]:=0;  //default
mb_Input_Registers[152]:=0;  //default
mb_Input_Registers[153]:=0;  //default
mb_Input_Registers[154]:=0;  //default
mb_Input_Registers[155]:=0;  //default
mb_Input_Registers[156]:=0;  //default
mb_Input_Registers[157]:=0;  //default
mb_Input_Registers[158]:=0;  //default
mb_Input_Registers[159]:=0;  //default
mb_Input_Registers[160]:=0;  //default
mb_Input_Registers[161]:=0;  //default
mb_Input_Registers[162]:=0;  //default
mb_Input_Registers[163]:=0;  //default
mb_Input_Registers[164]:=0;  //default
mb_Input_Registers[165]:=0;  //default
mb_Input_Registers[166]:=0;  //default
mb_Input_Registers[167]:=0;  //default
mb_Input_Registers[168]:=0;  //default
mb_Input_Registers[169]:=0;  //default
mb_Input_Registers[170]:=0;  //default
mb_Input_Registers[171]:=0;  //default
mb_Input_Registers[172]:=0;  //default
mb_Input_Registers[173]:=0;  //default
mb_Input_Registers[174]:=0;  //default
mb_Input_Registers[175]:=0;  //default
mb_Input_Registers[176]:=0;  //default
mb_Input_Registers[177]:=0;  //default
mb_Input_Registers[178]:=0;  //default
mb_Input_Registers[179]:=0;  //default
mb_Input_Registers[180]:=0;  //default
mb_Input_Registers[181]:=0;  //default
mb_Input_Registers[182]:=0;  //default
mb_Input_Registers[183]:=0;  //default
mb_Input_Registers[184]:=0;  //default
mb_Input_Registers[185]:=0;  //default
mb_Input_Registers[186]:=0;  //default
mb_Input_Registers[187]:=0;  //default
mb_Input_Registers[188]:=0;  //default
mb_Input_Registers[189]:=0;  //default
mb_Input_Registers[190]:=0;  //default
mb_Input_Registers[191]:=0;  //default
mb_Input_Registers[192]:=0;  //default
mb_Input_Registers[193]:=0;  //default
mb_Input_Registers[194]:=0;  //default
mb_Input_Registers[195]:=0;  //default
mb_Input_Registers[196]:=0;  //default
mb_Input_Registers[197]:=0;  //default
mb_Input_Registers[198]:=0;  //default
mb_Input_Registers[199]:=0;  //default
mb_Input_Registers[200]:=0;  //default
mb_Input_Registers[201]:=0;  //default
mb_Input_Registers[202]:=0;  //default
mb_Input_Registers[203]:=0;  //default
mb_Input_Registers[204]:=0;  //default
mb_Input_Registers[205]:=0;  //default
mb_Input_Registers[206]:=0;  //default
mb_Input_Registers[207]:=0;  //default
mb_Input_Registers[208]:=0;  //default
mb_Input_Registers[209]:=0;  //default
mb_Input_Registers[210]:=0;  //default
mb_Input_Registers[211]:=0;  //default
mb_Input_Registers[212]:=0;  //default
mb_Input_Registers[213]:=0;  //default
mb_Input_Registers[214]:=0;  //default
mb_Input_Registers[215]:=0;  //default
mb_Input_Registers[216]:=0;  //default
mb_Input_Registers[217]:=0;  //default
mb_Input_Registers[218]:=0;  //default
mb_Input_Registers[219]:=0;  //default
mb_Input_Registers[220]:=0;  //default
mb_Input_Registers[221]:=0;  //default
mb_Input_Registers[222]:=0;  //default
mb_Input_Registers[223]:=0;  //default
mb_Input_Registers[224]:=0;  //default
mb_Input_Registers[225]:=0;  //default
mb_Input_Registers[226]:=0;  //default
mb_Input_Registers[227]:=0;  //default
mb_Input_Registers[228]:=0;  //default
mb_Input_Registers[229]:=0;  //default
mb_Input_Registers[230]:=0;  //default
mb_Input_Registers[231]:=0;  //default
mb_Input_Registers[232]:=0;  //default
mb_Input_Registers[233]:=0;  //default
mb_Input_Registers[234]:=0;  //default
mb_Input_Registers[235]:=0;  //default
mb_Input_Registers[236]:=0;  //default
mb_Input_Registers[237]:=0;  //default
mb_Input_Registers[238]:=0;  //default
mb_Input_Registers[239]:=0;  //default
mb_Input_Registers[240]:=0;  //default
mb_Input_Registers[241]:=0;  //default
mb_Input_Registers[242]:=0;  //default
mb_Input_Registers[243]:=0;  //default
mb_Input_Registers[244]:=0;  //default
mb_Input_Registers[245]:=0;  //default
mb_Input_Registers[246]:=0;  //default
mb_Input_Registers[247]:=0;  //default
mb_Input_Registers[248]:=0;  //default
mb_Input_Registers[249]:=0;  //default
mb_Input_Registers[250]:=0;  //default
mb_Input_Registers[251]:=0;  //default
mb_Input_Registers[252]:=0;  //default
mb_Input_Registers[253]:=0;  //default
mb_Input_Registers[254]:=0;  //default
mb_Input_Registers[255]:=0;  //default

END_PROGRAM

// ---- POUs/Modbus/p_ModbusTx_PLCMemory.TcPOU
PROGRAM p_ModbusTx_PLCMemory
VAR
END_VAR

(* Send status information over modbus to IOC *)

(* The calculated effective radius *)
MEMCPY(destAddr:=ADR(mb_PLC_Memory[100]), srcAddr:=ADR(XRT_RADIUS), n:=SIZEOF(XRT_RADIUS));
MEMCPY(destAddr:=ADR(mb_PLC_Memory[102]), srcAddr:=ADR(TFS_RADIUS), n:=SIZEOF(TFS_RADIUS));

(* Individual lens radius *)
MEMCPY(destAddr:=ADR(mb_PLC_Memory[104]), srcAddr:=ADR(TFS_LENSES[1].RADIUS), n:=SIZEOF(TFS_LENSES[1].RADIUS));
MEMCPY(destAddr:=ADR(mb_PLC_Memory[106]), srcAddr:=ADR(TFS_LENSES[2].RADIUS), n:=SIZEOF(TFS_LENSES[2].RADIUS));
MEMCPY(destAddr:=ADR(mb_PLC_Memory[108]), srcAddr:=ADR(TFS_LENSES[3].RADIUS), n:=SIZEOF(TFS_LENSES[3].RADIUS));
MEMCPY(destAddr:=ADR(mb_PLC_Memory[110]), srcAddr:=ADR(TFS_LENSES[4].RADIUS), n:=SIZEOF(TFS_LENSES[4].RADIUS));
MEMCPY(destAddr:=ADR(mb_PLC_Memory[112]), srcAddr:=ADR(TFS_LENSES[5].RADIUS), n:=SIZEOF(TFS_LENSES[5].RADIUS));
MEMCPY(destAddr:=ADR(mb_PLC_Memory[114]), srcAddr:=ADR(TFS_LENSES[6].RADIUS), n:=SIZEOF(TFS_LENSES[6].RADIUS));
MEMCPY(destAddr:=ADR(mb_PLC_Memory[116]), srcAddr:=ADR(TFS_LENSES[7].RADIUS), n:=SIZEOF(TFS_LENSES[7].RADIUS));
MEMCPY(destAddr:=ADR(mb_PLC_Memory[118]), srcAddr:=ADR(TFS_LENSES[8].RADIUS), n:=SIZEOF(TFS_LENSES[8].RADIUS));
MEMCPY(destAddr:=ADR(mb_PLC_Memory[120]), srcAddr:=ADR(TFS_LENSES[9].RADIUS),  n:=SIZEOF(TFS_LENSES[9].RADIUS));
MEMCPY(destAddr:=ADR(mb_PLC_Memory[122]), srcAddr:=ADR(TFS_LENSES[10].RADIUS), n:=SIZEOF(TFS_LENSES[10].RADIUS));
MEMCPY(destAddr:=ADR(mb_PLC_Memory[124]), srcAddr:=ADR(XRT_LENSES[1].RADIUS), n:=SIZEOF(XRT_LENSES[1].RADIUS));
MEMCPY(destAddr:=ADR(mb_PLC_Memory[126]), srcAddr:=ADR(XRT_LENSES[2].RADIUS), n:=SIZEOF(XRT_LENSES[2].RADIUS));
MEMCPY(destAddr:=ADR(mb_PLC_Memory[128]), srcAddr:=ADR(XRT_LENSES[3].RADIUS), n:=SIZEOF(XRT_LENSES[3].RADIUS));

MEMCPY(destAddr:=ADR(mb_PLC_Memory[130]), srcAddr:=ADR(q_stActiveLimit.TRIP_LOW), n:=SIZEOF(q_stActiveLimit.TRIP_LOW));
MEMCPY(destAddr:=ADR(mb_PLC_Memory[132]), srcAddr:=ADR(q_stActiveLimit.TRIP_HIGH), n:=SIZEOF(q_stActiveLimit.TRIP_HIGH));

// MEMCPY(destAddr:=ADR(mb_PLC_Memory[134]), srcAddr:=ADR(iCycleCount), n:=SIZEOF(iCycleCount));
// Abuse the FLOAT port to send along 16-bit cycle information:
mb_PLC_Memory[134] := iCycleCount;
mb_PLC_Memory[135] := 0;

MEMCPY(destAddr:=ADR(mb_PLC_Memory[136]), srcAddr:=ADR(i_fPhotonEnergy), n:=SIZEOF(i_fPhotonEnergy));
// 137 taken up by fPhotonEnergy

(* Online/active values *)
mb_PLC_Memory[138]:=BOOL_TO_WORD(bHeartbeatAlive);
mb_PLC_Memory[139]:=BOOL_TO_WORD(bFAULT);
mb_PLC_Memory[140]:=BOOL_TO_WORD(bStateFault);
mb_PLC_Memory[141]:=BOOL_TO_WORD(bLimitSummaryFault);
mb_PLC_Memory[142]:=BOOL_TO_WORD(bMinEnergyFault);
mb_PLC_Memory[143]:=BOOL_TO_WORD(bRequiresTransfocatorFault);
mb_PLC_Memory[144]:=BOOL_TO_WORD(bTableLimitFault);
mb_PLC_Memory[145]:=BOOL_TO_WORD(FALSE);
mb_PLC_Memory[146]:=BOOL_TO_WORD(FALSE);
mb_PLC_Memory[147]:=BOOL_TO_WORD(FALSE);

(* Latched fault information *)
mb_PLC_Memory[148]:=BOOL_TO_WORD(q_bHeartbeatLatch);
mb_PLC_Memory[149]:=BOOL_TO_WORD(q_bFaultLatch);
mb_PLC_Memory[150]:=BOOL_TO_WORD(q_bStateLatch);
mb_PLC_Memory[151]:=BOOL_TO_WORD(q_bLimitSummaryFaultLatch);
mb_PLC_Memory[152]:=BOOL_TO_WORD(q_bMinEnergyFaultLatch);
mb_PLC_Memory[153]:=BOOL_TO_WORD(q_bRequiresTransfocatorFaultLatch);
mb_PLC_Memory[154]:=BOOL_TO_WORD(q_bTableLimitFaultLatch);
mb_PLC_Memory[155]:=BOOL_TO_WORD(FALSE);
mb_PLC_Memory[156]:=BOOL_TO_WORD(FALSE);
mb_PLC_Memory[157]:=BOOL_TO_WORD(FALSE);

END_PROGRAM

// ---- POUs/FB_EnergyTables.TcPOU

(* WARNING: This file is auto-generated. Do not modify it.*)
FUNCTION_BLOCK FB_EnergyTables
VAR_INPUT
END_VAR
VAR_OUTPUT
    stNO_LENS : ARRAY[0..978] OF ST_TableRow;
	stLENS3_333 : ARRAY[0..665] OF ST_TableRow;
	stLENS2_428 : ARRAY[0..734] OF ST_TableRow;
	stLENS1_750 : ARRAY[0..898] OF ST_TableRow;
END_VAR
VAR
    bInitialized : BOOL := FALSE;
END_VAR


(* WARNING: This file is auto-generated. Do not modify it.*)
IF NOT bInitialized THEN
    
